PROGRAM ControlPanel
VAR
	
	IsProductLeavingTrig: F_TRIG;
	EmergencyTilt: TON;
END_VAR

IsProductLeavingTrig(CLK:=gvl.IsProductLeaving , Q=> );
CASE gvl.CurrentControlPanelState OF 
	
	ControlPanelStates.WaitingToStart:
	
	gvl.StopLight:=FALSE;
	gvl.StartLight:=FALSE;
	gvl.ResetLight:=FALSE;
	IF GVL.Start  THEN	
	gvl.CurrentBaseState:=BaseStates.LocatingBaseInPlace;
	gvl.CurrentLidsState:=LidStates.LocatingInPlace;
	gvl.CurrentRobotState:=ManipulatorStates.WaitingForALid;
	gvl.CurrentControlPanelState:=ControlPanelStates.Working;				
		ELSIF NOT gvl.Stop  THEN
			gvl.CurrentControlPanelState:=ControlPanelStates.Stopping;
		ELSIF NOT gvl.EmergencyStop THEN
			gvl.CurrentControlPanelState:=ControlPanelStates.Emergency;
	END_IF
	
	ControlPanelStates.Working:
	gvl.ResetAfterEmergency:=FALSE;
	gvl.StopLight:=FALSE;
	gvl.StartLight:=TRUE;
	IF gvl.CountReset THEN
		gvl.ResetLight:=TRUE;
	END_IF
	gvl.ResetLight:=FALSE;	
	IF NOT gvl.Stop  THEN
			gvl.CurrentControlPanelState:=ControlPanelStates.Stopping;
		ELSIF NOT gvl.EmergencyStop THEN
			gvl.CurrentControlPanelState:=ControlPanelStates.Emergency;	
	END_IF
	
	ControlPanelStates.Stopping:
	
	IF IsProductLeavingTrig.Q THEN
		gvl.CurrentBaseState:=BaseStates.Stop;
		gvl.CurrentLidsState:=LidStates.Stop;
		gvl.CurrentRobotState:=ManipulatorStates.Stop;
	ELSE
		// Waits for the product to be finished
	END_IF
	gvl.StartLight:=FALSE;
	gvl.StopLight:=TRUE;
	IF gvl.Start THEN
		gvl.CurrentBaseState:=BaseStates.LocatingBaseInPlace;
		gvl.CurrentLidsState:=LidStates.LocatingInPlace;
		gvl.CurrentRobotState:=ManipulatorStates.WaitingForALid;
		gvl.CurrentControlPanelState:=ControlPanelStates.Working;	
		ELSIF not gvl.EmergencyStop THEN
			gvl.CurrentControlPanelState:=ControlPanelStates.Emergency;	
	END_IF
	
	ControlPanelStates.Emergency:
	
	gvl.CurrentBaseState:=BaseStates.Stop;
	gvl.CurrentLidsState:=LidStates.Stop;
	gvl.CurrentRobotState:=ManipulatorStates.Stop;
	gvl.StartLight:=FALSE;
	EmergencyTilt(IN:=NOT EmergencyTilt.Q , PT:=T#0.5S , Q=>gvl.StopLight , ET=> );
	IF gvl.Start AND gvl.EmergencyStop THEN
		gvl.CurrentBaseState:=BaseStates.LocatingBaseInPlace;
		gvl.CurrentLidsState:=LidStates.LocatingInPlace;
		gvl.CurrentRobotState:=ManipulatorStates.WaitingForALid;
		gvl.CurrentControlPanelState:=ControlPanelStates.Working;
		gvl.ResetAfterEmergency:=TRUE;
	END_IF
		
END_CASE

END_PROGRAM

(* stored: Version 1.1.0.1, ProductVersion 3.1.4024.9
   POU ControlPanel: Id {d293cf6d-ff19-47fe-b382-d19e3c745654}, SpecialFunc None *)
